{attribute 'GeneratedUsingTerminal: '}
{attribute addProperty BoxType ""}
{attribute addProperty Id "unreferencedAT %I*SyncUnitTask_2D604ED59PlcTaskAT %I*SyncUnitTask_2D604ED59"}
{attribute addProperty CRC "1877705303"}
{attribute addProperty Size "18"}
TYPE SyncUnitTasks_6FEB8257 :
STRUCT
	{attribute addProperty Name "unreferenced"}
	unreferenced : TcoIo.SyncUnitTask_2D604ED5;
	{attribute addProperty Name "PlcTask"}
	PlcTask : TcoIo.SyncUnitTask_2D604ED5;
END_STRUCT
END_TYPE

(* stored: Version 1.2.0.0, ProductVersion 3.1.4024.9
   DUT SyncUnitTasks_6FEB8257: Id {65fa2c96-6f19-4084-9422-7bd61560c813} *)
